// TIA Portal V18 export
DATA_BLOCK "not_used_blocks_DB"   // DB68
VERSION : 0.1
// stored: AutoNumber true, DBAccessibleFromOPCUA true, InstanceOfName not_used_blocks, InstanceOfType FB
"not_used_blocks"
   // VAR
   //    isMultiturn : Bool;
   //    MultiTurnGoesFwdOnly : Bool;
   //    SET_SPD_ABS : Real;
   //    POS : Real;
   //    TARGET : Real;
   //    par_lim_fwd : Real;
   //    par_lim_rev : Real;
   //    par_spd_absmax : Real;
   //    par_dist_absMax : Real;
   //    par_spd_crawl : Real;
   //    par_dist_crawl : Real;
   //    par_dist_stop : Real;
   //    speed_limited_by_target : Real;
   //    ER : Bool;
   //    ER_w : WString;
   //    mot_universal_arrived_missed_Instance { S7_SetPoint := 'True'} : "mot_universal_arrived_missed";
   //    was_set : Bool;
   // END_VAR
BEGIN
END_DATA_BLOCK
